FUNCTION transform : ST_Frame
VAR_IN_OUT CONSTANT
	i_frame1 :ST_Frame;
	i_frame2 :ST_Frame;
END_VAR
VAR
END_VAR

transform.m_rot := mat3Mat3(i_frame1.m_rot, i_frame2.m_rot);
transform.m_pos := mat3Vec3(i_frame1.m_rot, i_frame2.m_pos);
transform.m_pos :=addVec3(transform.m_pos,i_frame1.m_pos);

END_FUNCTION

(* stored: Version 1.1.0.1, ProductVersion 3.1.4024.12
   POU transform: Id {7ca6f97b-de44-4b21-a77a-278a6c7df5be}, SpecialFunc None *)
